Staubli VAL3: moveOffside.pgx

program moveOffside()
begin
  movej(parkingPosition,flange,mFastMov)
  waitEndMove()
  message="moveOffside:done"
  taskCreate "sendStatus",100,sendStatus()
  taskKill("moveOffside")
end
